TYPE Robot_FW :
	
STRUCT
	FW_Version :DINT;
	FW_Major:DINT;
	FW_Minor:DINT;
	
END_STRUCT


END_TYPE

(* stored: Version 1.1.0.1, ProductVersion 3.1.4024.10
   DUT Robot_FW: Id {725a0fad-23e5-4548-aada-d6d381166096} *)
